{attribute addProperty BoxType "EL1054-0000-0016"}
{attribute addProperty Id "ChannelAT %I*ARRAY[0..6] OF Channel_E18390666480WcStateAT %I*WcState_98A4DF7520.250InfoDataAT %I*InfoData_192954DE1620"}
{attribute addProperty CRC "3462302143"}
{attribute addProperty SizeInBites "82"}
{attribute addProperty SizeInBytes "10.25"}
TYPE EL1054_27203488 :
STRUCT
	{attribute addProperty Name "Channel"}
	Channel : ARRAY[0..6] OF Channel_E1839066;
	{attribute addProperty Name "WcState"}
	WcState : WcState_98A4DF75;
	{attribute addProperty Name "InfoData"}
	InfoData : InfoData_192954DE;
END_STRUCT
END_TYPE

(* stored: Version 1.2.0.0, ProductVersion 3.1.4024.9
   DUT EL1054_27203488: Id {cc456ccd-c8cd-46ef-bff2-606626d87dee} *)
